(* IEC 61131-3 sources: LogicCraft_ABB/, 1 file *)

(* ---- test.st ---- *)
PROGRAM SimpleTest
VAR
    x : INT := 0;
END_VAR

x := x + 1;
END_PROGRAM
